// TIA Portal V20 export
TYPE "typeEstopElement"
// stored: Access Published, IsFailsafeCompliant true, Namespace Safety
   STRUCT
      EstopE0 : Bool;   // OP PANEL NoPress Estop
      EstopE1 : Bool;   // NoPress Estop01
      EstopE2 : Bool;   // NoPress Estop02
      EstopE3 : Bool;   // NoPress Estop03
      EstopE4 : Bool;   // NoPress Estop04
      EstopE5 : Bool;   // NoPress Estop05
      EstopE6 : Bool;   // NoPress Estop06
      EstopE7 : Bool;   // NoPress Estop07
      EstopE8 : Bool;   // NoPress Estop08
      EstopE9 : Bool;   // NoPress Estop09
      EstopE10 : Bool;   // NoPress Estop10
   END_STRUCT;
END_TYPE
